{attribute addProperty BoxType "EK1122-0000-0018"}
{attribute addProperty Id "Beckhoff_ER5xxxsub_EK1100EK1100_179A0949162A_0001_ER5101_0002_0019ER5101_F338D8E417622A_0002_ER5101_1002_0017ER5101_F338D8E417622A_0003_ER5151_0002_0018ER5151_BA9EF92517622"}
{attribute addProperty CRC "4012526237"}
{attribute addProperty SizeInBites "544"}
{attribute addProperty SizeInBytes "68"}
TYPE Beckhoff_ER5xxxEK1122_EF2A4A9D EXTENDS EK1122_179A0949 :
STRUCT
	{attribute addProperty Name "Beckhoff_ER5xxxsub_EK1100"}
	Beckhoff_ER5xxxsub_EK1100 : EK1100_179A0949;
	{attribute addProperty Name "A_0001_ER5101_0002_0019"}
	A_0001_ER5101_0002_0019 : ER5101_F338D8E4;
	{attribute addProperty Name "A_0002_ER5101_1002_0017"}
	A_0002_ER5101_1002_0017 : ER5101_F338D8E4;
	{attribute addProperty Name "A_0003_ER5151_0002_0018"}
	A_0003_ER5151_0002_0018 : ER5151_BA9EF925;
END_STRUCT
END_TYPE

(* stored: Version 1.2.0.0, ProductVersion 3.1.4024.9
   DUT Beckhoff_ER5xxxEK1122_EF2A4A9D: Id {2bd91da4-926f-42f9-868d-8f6524551a0f} *)
